(* Schneider Machine Expert - Basic project m5, file version 2.0.0.0 *)
(* ProjectInformations: Name=New project *)

HARDWARE
  Cpu 0: TM221CE16R
  EthernetConfiguration: NetworkName=M221, IpAllocationMode=FixedAddress, IpAddress=0.0.0.0, SubnetMask=0.0.0.0
  SerialLineConfiguration: Baud=Baud19200, Parity=ParityEven, DataBits=DataBits8, StopBits=StopBits1, PhysicalMedium=PhysicalMediumRs485, TransmissionMode=TransmissionModeModbusRtu, SlaveId=1, Addressing=SlaveAddressing
  MastTask: UsePeriodScanMode=false, PeriodScan=100
  FastTask: Period=255
  CpuBehavior: StartingMode=StartAsPreviousState, AutoSaveRamOnEeprom=true, WatchdogPeriod=250

SYMBOLS  (address, symbol, comment, settings)

POU New POU
  (* SectionNumber=1 *)

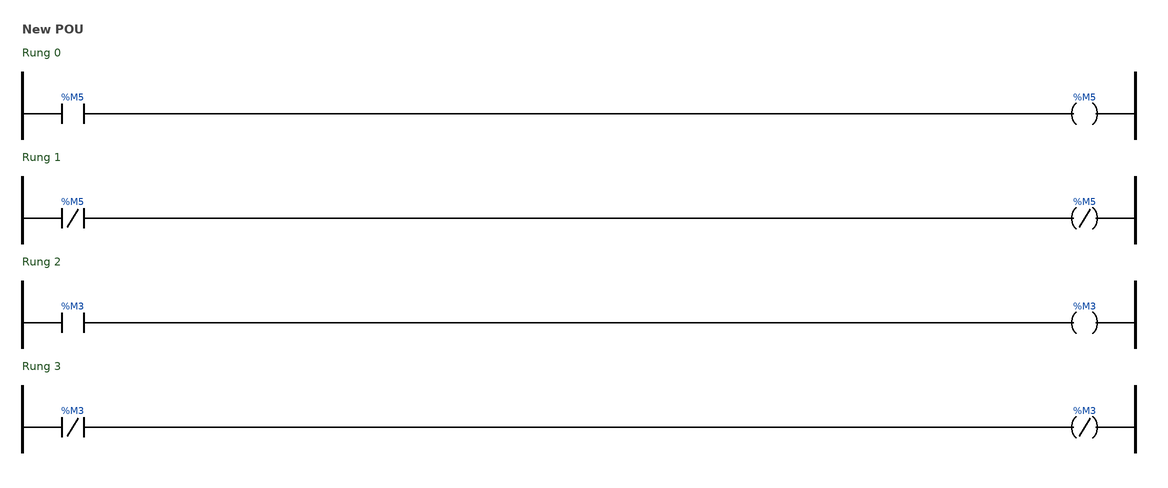

// Rung 0
  LD %M5
  ST %M5
  // as ST:
  //   %M5 := %M5;

// Rung 1
  LDN %M5
  STN %M5
  // as ST:
  //   %M5 := NOT (NOT %M5);

// Rung 2
  LD %M3
  ST %M3
  // as ST:
  //   %M3 := %M3;

// Rung 3
  LDN %M3
  STN %M3
  // as ST:
  //   %M3 := NOT (NOT %M3);
